Staubli VAL3: loopReadForce.pgx

public program loopReadForce(num& x_nSensorForce[], FlagStatus& x_fSensorStatus)
  local num l_nDetectValue[6]
begin

  //This program is used for circularly acquiring the interaction force/torque values between the robot endeffector and environment.

  //do
  //Acquire the detected values from the sensor
  call readDetectValue(l_nDetectValue,x_fSensorStatus)
  //Calculate the sensor force/torque values
  call calculateForce(l_nDetectValue,x_nSensorForce)
  //until false

end
